TYPE ST_SPM_HMI_03_Alarmy_DaneElementuOZadanymIDZgloszenia :
STRUCT
	uiIDElementu				: UINT;
	sKodElementu				: STRING;
	sRodzajZgloszenia			: STRING;
	eRodzajZgloszenia			: B_Baza.E_Zgloszenia_Rodzaj;
	wsOpis						: WSTRING;
	wsTekstElementu				: WSTRING;
END_STRUCT
END_TYPE

(* stored: Version 1.1.0.1
   DUT ST_SPM_HMI_03_Alarmy_DaneElementuOZadanymIDZgloszenia: Id {64770227-c5a3-0033-2695-7c134f0dbfad} *)
